Xinje XDPPro project, PLC1: XD5E-60T10 (software 3.5.3 2018-11-19)

PROGRAM Ladder

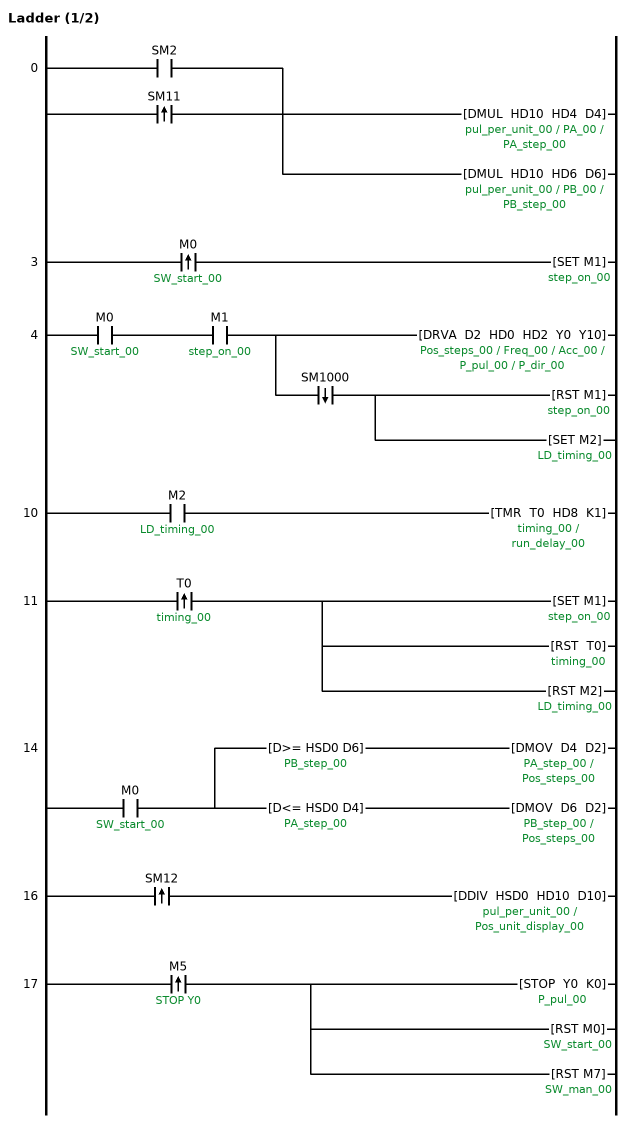
LD     SM2
ORP    SM11
DMUL   HD10 HD4 D4	; pul_per_unit_00 / PA_00 / PA_step_00
DMUL   HD10 HD6 D6	; pul_per_unit_00 / PB_00 / PB_step_00
LDP    M0	; SW_start_00
SET    M1	; step_on_00
LD     M0	; SW_start_00
AND    M1	; step_on_00
DRVA   D2 HD0 HD2 Y0 Y10	; Pos_steps_00 / Freq_00 / Acc_00 / P_pul_00 / P_dir_00
ANDF   SM1000
RST    M1	; step_on_00
SET    M2	; LD_timing_00
LD     M2	; LD_timing_00
TMR    T0 HD8 K1	; timing_00 / run_delay_00
LDP    T0	; timing_00
SET    M1	; step_on_00
RST    T0	; timing_00
RST    M2	; LD_timing_00
LD     M0	; SW_start_00
MPS
DAND>= HSD0 D6	; PB_step_00
DMOV   D4 D2	; PA_step_00 / Pos_steps_00
MPP
DAND<= HSD0 D4	; PA_step_00
DMOV   D6 D2	; PB_step_00 / Pos_steps_00
LDP    SM12
DDIV   HSD0 HD10 D10	; pul_per_unit_00 / Pos_unit_display_00
LDP    M5	; STOP Y0
STOP   Y0 K0	; P_pul_00
RST    M0	; SW_start_00
RST    M7	; SW_man_00

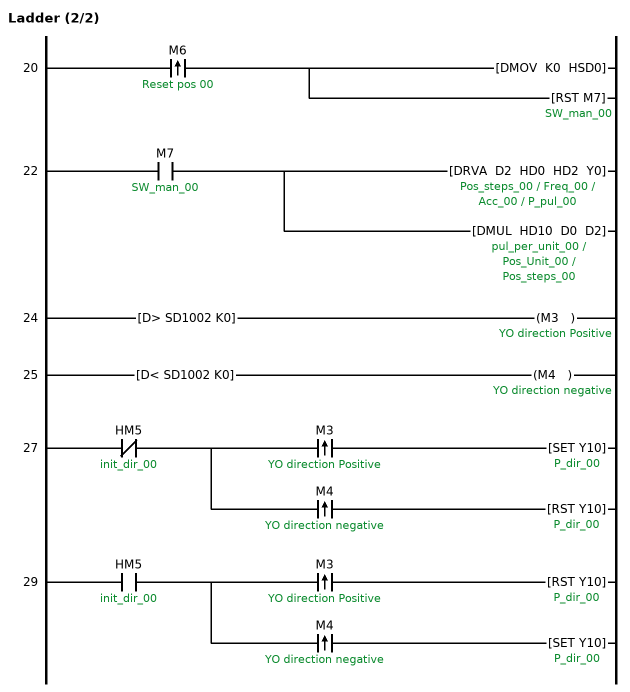
LDP    M6	; Reset pos 00
DMOV   K0 HSD0
RST    M7	; SW_man_00
LD     M7	; SW_man_00
DRVA   D2 HD0 HD2 Y0	; Pos_steps_00 / Freq_00 / Acc_00 / P_pul_00
DMUL   HD10 D0 D2	; pul_per_unit_00 / Pos_Unit_00 / Pos_steps_00
DLD>   SD1002 K0
OUT    M3	; YO direction Positive
DLD<   SD1002 K0
OUT    M4	; YO direction negative
LDI    HM5	; init_dir_00
MPS
ANDP   M3	; YO direction Positive
SET    Y10	; P_dir_00
MPP
ANDP   M4	; YO direction negative
RST    Y10	; P_dir_00
LD     HM5	; init_dir_00
MPS
ANDP   M3	; YO direction Positive
RST    Y10	; P_dir_00
MPP
ANDP   M4	; YO direction negative
SET    Y10	; P_dir_00

COMMENTS (devices not used above)
Y1	P-pul_01
Y7	Chieu01
Y11	P_dir_01
M100	SW_start_00
M101	step_on_00
M102	LD_timing_00
M103	YO direction Positive
M104	YO direction negative
M105	STOP Y0
M106	Reset pos 00
M110	SW_start_01
D110	Pos_steps_01
D202	Pos 01
D204	Tan so 01
D206	Gia toc 01
HD100	Freq_00
HD102	Acc_00
HD104	PA_00
HD106	PB_00
HD108	run_delay_00
HD110	pul_per_unit_00
HD200	Step_per_unit_00